// Settings for GreenMaster
TYPE RedundancySettings :
STRUCT
B_AMSID:STRING;		// AMS-ID Redundant aggregat
B_VARIABLE:STRING;	
END_STRUCT
END_TYPE

(* stored: Version 1.1.0.1, ProductVersion 3.1.4024.6
   DUT RedundancySettings: Id {a6785c38-8e5a-4fbd-aa09-b6c5721ce1cb} *)
